LIN {X 0,Y 239.218,Z 1199.48,A -85,B 0,C 180,E1 5752.201,E2 5752.201} C_VEL
LIN {X 0,Y 256.307,Z 1187.286,A -85,B 0,C 180,E1 5754.218,E2 5754.218} C_VEL
LIN {X 0,Y 273.673,Z 1173.769,A -85,B 0,C 180,E1 5755.98,E2 5755.98} C_VEL
LIN {X 0,Y 294.221,Z 1156.22,A -85,B 0,C 180,E1 5757.756,E2 5757.756} C_VEL
LIN {X 0,Y 314.021,Z 1137.067,A -85,B 0,C 180,E1 5759.227,E2 5759.227} C_VEL
LIN {X 0,Y 329.492,Z 1120.573,A -85,B 0,C 180,E1 5760.229,E2 5760.229} C_VEL
LIN {X 0,Y 333.53,Z 1116.052,A -85,B 0,C 180,E1 5760.492,E2 5760.492} C_VEL
LIN {X 0,Y 325.823,Z 1124.556,A -85,B 0,C 180,E1 5761.006,E2 5761.006} C_VEL
LIN {X 0,Y 321.322,Z 1129.417,A -85,B 0,C 180,E1 5761.15,E2 5761.15} C_VEL
LIN {X 0,Y 315.113,Z 1135.776,A -85,B 0,C 180,E1 5760.961,E2 5760.961} C_VEL
LIN {X 0,Y 300.81,Z 1149.589,A -85,B 0,C 180,E1 5759.861,E2 5759.861} C_VEL
LIN {X 0,Y 283.612,Z 1164.923,A -85,B 0,C 180,E1 5758.586,E2 5758.586} C_VEL
LIN {X 0,Y 260.469,Z 1183.452,A -85,B 0,C 180,E1 5756.565,E2 5756.565} C_VEL
LIN {X 0,Y 240.904,Z 1197.395,A -85,B 0,C 180,E1 5754.522,E2 5754.522} C_VEL
LIN {X 0,Y 222.759,Z 1209.185,A -85,B 0,C 180,E1 5752.261,E2 5752.261} C_VEL
LIN {X 0,Y 204.429,Z 1220.07,A -85,B 0,C 180,E1 5749.508,E2 5749.508} C_VEL
LIN {X 0,Y 182.016,Z 1232.203,A -85,B 0,C 180,E1 5745.247,E2 5745.247} C_VEL
LIN {X 0,Y 160.819,Z 1242.295,A -85,B 0,C 180,E1 5739.896,E2 5739.896} C_VEL
LIN {X 0,Y 143.477,Z 1249.877,A -85,B 0,C 180,E1 5733.957,E2 5733.957} C_VEL
LIN {X 0,Y 128.105,Z 1256.155,A -85,B 0,C 180,E1 5726.665,E2 5726.665} C_VEL
LIN {X 0,Y 112.467,Z 1262.354,A -85,B 0,C 180,E1 5715.366,E2 5715.366} C_VEL
LIN {X 0,Y 101.995,Z 1266.473,A -85,B 0,C 180,E1 5701.992,E2 5701.992} C_VEL
LIN {X 0,Y 97.397,Z 1268.698,A -85,B 0,C 180,E1 5689.83,E2 5689.83} C_VEL
LIN {X 0,Y 96.077,Z 1269.823,A -85,B 0,C 180,E1 5678.405,E2 5678.405} C_VEL
LIN {X 0,Y 96.068,Z 1270.167,A -85,B 0,C 180,E1 5670.027,E2 5670.027} C_VEL
LIN {X 0,Y 96.076,Z 1269.821,A -85,B 0,C 180,E1 5661.65,E2 5661.65} C_VEL
LIN {X 0,Y 97.385,Z 1268.69,A -85,B 0,C 180,E1 5650.225,E2 5650.225} C_VEL
LIN {X 0,Y 102.276,Z 1266.336,A -85,B 0,C 180,E1 5637.505,E2 5637.505} C_VEL
LIN {X 0,Y 114.151,Z 1261.596,A -85,B 0,C 180,E1 5623.097,E2 5623.097} C_VEL
LIN {X 0,Y 128.042,Z 1256.122,A -85,B 0,C 180,E1 5613.367,E2 5613.367} C_VEL
LIN {X 0,Y 142.747,Z 1250.113,A -85,B 0,C 180,E1 5606.335,E2 5606.335} C_VEL
LIN {X 0,Y 159.123,Z 1242.966,A -85,B 0,C 180,E1 5600.603,E2 5600.603} C_VEL
LIN {X 0,Y 178.447,Z 1233.818,A -85,B 0,C 180,E1 5595.538,E2 5595.538} C_VEL
LIN {X 0,Y 202.513,Z 1221.049,A -85,B 0,C 180,E1 5590.808,E2 5590.808} C_VEL
LIN {X 0,Y 221.991,Z 1209.52,A -85,B 0,C 180,E1 5587.838,E2 5587.838} C_VEL
LIN {X 0,Y 240.822,Z 1197.285,A -85,B 0,C 180,E1 5585.48,E2 5585.48} C_VEL
LIN {X 0,Y 262.332,Z 1181.904,A -85,B 0,C 180,E1 5583.249,E2 5583.249} C_VEL
LIN {X 0,Y 283.988,Z 1164.363,A -85,B 0,C 180,E1 5581.374,E2 5581.374} C_VEL
LIN {X 0,Y 300.904,Z 1149.241,A -85,B 0,C 180,E1 5580.123,E2 5580.123} C_VEL
LIN {X 0,Y 311.366,Z 1139.22,A -85,B 0,C 180,E1 5579.418,E2 5579.418} C_VEL
LIN {X 0,Y 289.81,Z 1158.959,A -85,B 0,C 180,E1 5577.825,E2 5577.825} C_VEL
LIN {X 0,Y 272.462,Z 1173.195,A -85,B 0,C 180,E1 5576.347,E2 5576.347} C_VEL
LIN {X 0,Y 255.986,Z 1185.54,A -85,B 0,C 180,E1 5574.748,E2 5574.748} C_VEL
LIN {X 0,Y 238.263,Z 1197.663,A -85,B 0,C 180,E1 5572.767,E2 5572.767} C_VEL
LIN {X 0,Y 217.251,Z 1210.706,A -85,B 0,C 180,E1 5569.951,E2 5569.951} C_VEL
LIN {X 0,Y 194.579,Z 1223.116,A -85,B 0,C 180,E1 5566.15,E2 5566.15} C_VEL
LIN {X 0,Y 176.306,Z 1232.089,A -85,B 0,C 180,E1 5562.263,E2 5562.263} C_VEL
LIN {X 0,Y 158.961,Z 1239.833,A -85,B 0,C 180,E1 5557.565,E2 5557.565} C_VEL
LIN {X 0,Y 142.135,Z 1246.704,A -85,B 0,C 180,E1 5551.519,E2 5551.519} C_VEL
LIN {X 0,Y 123.389,Z 1253.713,A -85,B 0,C 180,E1 5541.779,E2 5541.779} C_VEL
LIN {X 0,Y 110.564,Z 1258.126,A -85,B 0,C 180,E1 5531.279,E2 5531.279} C_VEL
LIN {X 0,Y 102.223,Z 1261.043,A -85,B 0,C 180,E1 5519.893,E2 5519.893} C_VEL
LIN {X 0,Y 97.807,Z 1262.768,A -85,B 0,C 180,E1 5508.447,E2 5508.447} C_VEL
LIN {X 0,Y 96.278,Z 1263.591,A -85,B 0,C 180,E1 5497.731,E2 5497.731} C_VEL
LIN {X 0,Y 96.072,Z 1263.825,A -85,B 0,C 180,E1 5488.78,E2 5488.78} C_VEL
LIN {X 0,Y 96.5,Z 1263.503,A -85,B 0,C 180,E1 5479.224,E2 5479.224} C_VEL
LIN {X 0,Y 99.61,Z 1262.139,A -85,B 0,C 180,E1 5465.67,E2 5465.67} C_VEL
LIN {X 0,Y 107.516,Z 1259.227,A -85,B 0,C 180,E1 5452.107,E2 5452.107} C_VEL
LIN {X 0,Y 118.163,Z 1255.541,A -85,B 0,C 180,E1 5441.841,E2 5441.841} C_VEL
LIN {X 0,Y 130.982,Z 1250.967,A -85,B 0,C 180,E1 5433.656,E2 5433.656} C_VEL
LIN {X 0,Y 146.56,Z 1245.028,A -85,B 0,C 180,E1 5426.621,E2 5426.621} C_VEL
LIN {X 0,Y 167.103,Z 1236.5,A -85,B 0,C 180,E1 5420.007,E2 5420.007} C_VEL
LIN {X 0,Y 188.41,Z 1226.357,A -85,B 0,C 180,E1 5414.971,E2 5414.971} C_VEL
LIN {X 0,Y 207.193,Z 1216.475,A -85,B 0,C 180,E1 5411.532,E2 5411.532} C_VEL
LIN {X 0,Y 225.646,Z 1205.779,A -85,B 0,C 180,E1 5408.77,E2 5408.77} C_VEL
LIN {X 0,Y 248.133,Z 1191.364,A -85,B 0,C 180,E1 5406.014,E2 5406.014} C_VEL
LIN {X 0,Y 269.668,Z 1175.589,A -85,B 0,C 180,E1 5403.827,E2 5403.827} C_VEL
LIN {X 0,Y 286.244,Z 1162.22,A -85,B 0,C 180,E1 5402.382,E2 5402.382} C_VEL
LIN {X 0,Y 303.049,Z 1147.355,A -85,B 0,C 180,E1 5401.092,E2 5401.092} C_VEL
LIN {X 0,Y 310.756,Z 1140.13,A -85,B 0,C 180,E1 5400.53,E2 5400.53} C_VEL
LIN {X 0,Y 300.81,Z 1149.589,A -85,B 0,C 180,E1 5399.861,E2 5399.861} C_VEL
LIN {X 0,Y 295.137,Z 1154.893,A -85,B 0,C 180,E1 5399.66,E2 5399.66} C_VEL
LIN {X 0,Y 278.947,Z 1168.594,A -85,B 0,C 180,E1 5399.771,E2 5399.771} C_VEL
LIN {X 0,Y 273.814,Z 1172.595,A -85,B 0,C 180,E1 5399.544,E2 5399.544} C_VEL
LIN {X 0,Y 256.149,Z 1186.028,A -85,B 0,C 180,E1 5398.058,E2 5398.058} C_VEL
LIN {X 0,Y 238.493,Z 1198.284,A -85,B 0,C 180,E1 5396.336,E2 5396.336} C_VEL
LIN {X 0,Y 219.173,Z 1210.502,A -85,B 0,C 180,E1 5394.09,E2 5394.09} C_VEL
LIN {X 0,Y 195.602,Z 1223.934,A -85,B 0,C 180,E1 5390.668,E2 5390.668} C_VEL
LIN {X 0,Y 173.778,Z 1234.85,A -85,B 0,C 180,E1 5386.557,E2 5386.557} C_VEL
LIN {X 0,Y 155.3,Z 1243.23,A -85,B 0,C 180,E1 5381.998,E2 5381.998} C_VEL
LIN {X 0,Y 137.722,Z 1250.508,A -85,B 0,C 180,E1 5376.215,E2 5376.215} C_VEL
LIN {X 0,Y 118.244,Z 1257.965,A -85,B 0,C 180,E1 5366.877,E2 5366.877} C_VEL
LIN {X 0,Y 103.112,Z 1263.274,A -85,B 0,C 180,E1 5355.096,E2 5355.096} C_VEL
LIN {X 0,Y 94.07,Z 1266.568,A -85,B 0,C 180,E1 5342.857,E2 5342.857} C_VEL
LIN {X 0,Y 89.575,Z 1268.504,A -85,B 0,C 180,E1 5330.958,E2 5330.958} C_VEL
LIN {X 0,Y 88.096,Z 1269.562,A -85,B 0,C 180,E1 5319.084,E2 5319.084} C_VEL
LIN {X 0,Y 88.065,Z 1269.889,A -85,B 0,C 180,E1 5310.68,E2 5310.68} C_VEL
LIN {X 0,Y 88.074,Z 1269.61,A -85,B 0,C 180,E1 5302.2,E2 5302.2} C_VEL
LIN {X 0,Y 89.152,Z 1268.721,A -85,B 0,C 180,E1 5291.051,E2 5291.051} C_VEL
LIN {X 0,Y 93.127,Z 1266.92,A -85,B 0,C 180,E1 5279.013,E2 5279.013} C_VEL
LIN {X 0,Y 101.184,Z 1263.918,A -85,B 0,C 180,E1 5266.992,E2 5266.992} C_VEL
LIN {X 0,Y 113.098,Z 1259.676,A -85,B 0,C 180,E1 5256.479,E2 5256.479} C_VEL
LIN {X 0,Y 128.614,Z 1253.989,A -85,B 0,C 180,E1 5247.641,E2 5247.641} C_VEL
LIN {X 0,Y 151.313,Z 1244.882,A -85,B 0,C 180,E1 5239.161,E2 5239.161} C_VEL
LIN {X 0,Y 170.149,Z 1236.454,A -85,B 0,C 180,E1 5234.233,E2 5234.233} C_VEL
LIN {X 0,Y 188.136,Z 1227.63,A -85,B 0,C 180,E1 5230.605,E2 5230.605} C_VEL
LIN {X 0,Y 206.734,Z 1217.61,A -85,B 0,C 180,E1 5227.597,E2 5227.597} C_VEL
LIN {X 0,Y 229.667,Z 1203.974,A -85,B 0,C 180,E1 5224.637,E2 5224.637} C_VEL
LIN {X 0,Y 252.115,Z 1188.752,A -85,B 0,C 180,E1 5222.304,E2 5222.304} C_VEL
LIN {X 0,Y 269.932,Z 1175.428,A -85,B 0,C 180,E1 5220.751,E2 5220.751} C_VEL
LIN {X 0,Y 286.918,Z 1161.515,A -85,B 0,C 180,E1 5219.471,E2 5219.471} C_VEL
LIN {X 0,Y 288.401,Z 1160.248,A -85,B 0,C 180,E1 5219.367,E2 5219.367} C_VEL
LIN {X 0,Y 271.073,Z 1174.227,A -85,B 0,C 180,E1 5218.002,E2 5218.002} C_VEL
LIN {X 0,Y 253.408,Z 1187.192,A -85,B 0,C 180,E1 5216.413,E2 5216.413} C_VEL
LIN {X 0,Y 232.122,Z 1201.336,A -85,B 0,C 180,E1 5214.155,E2 5214.155} C_VEL
LIN {X 0,Y 208.446,Z 1215.124,A -85,B 0,C 180,E1 5211.069,E2 5211.069} C_VEL
LIN {X 0,Y 190.022,Z 1224.734,A -85,B 0,C 180,E1 5208.077,E2 5208.077} C_VEL
LIN {X 0,Y 172.194,Z 1233.152,A -85,B 0,C 180,E1 5204.493,E2 5204.493} C_VEL
LIN {X 0,Y 153.483,Z 1241.135,A -85,B 0,C 180,E1 5199.678,E2 5199.678} C_VEL
LIN {X 0,Y 131.593,Z 1249.466,A -85,B 0,C 180,E1 5191.764,E2 5191.764} C_VEL
LIN {X 0,Y 115.247,Z 1254.97,A -85,B 0,C 180,E1 5182.916,E2 5182.916} C_VEL
LIN {X 0,Y 103.502,Z 1258.699,A -85,B 0,C 180,E1 5173.268,E2 5173.268} C_VEL
LIN {X 0,Y 94.868,Z 1261.418,A -85,B 0,C 180,E1 5161.768,E2 5161.768} C_VEL
LIN {X 0,Y 89.971,Z 1263.097,A -85,B 0,C 180,E1 5149.444,E2 5149.444} C_VEL
LIN {X 0,Y 88.322,Z 1263.854,A -85,B 0,C 180,E1 5138.433,E2 5138.433} C_VEL
LIN {X 0,Y 88.078,Z 1264.087,A -85,B 0,C 180,E1 5128.669,E2 5128.669} C_VEL
LIN {X 0,Y 88.591,Z 1263.768,A -85,B 0,C 180,E1 5118.249,E2 5118.249} C_VEL
LIN {X 0,Y 92.226,Z 1262.407,A -85,B 0,C 180,E1 5103.578,E2 5103.578} C_VEL
LIN {X 0,Y 101.128,Z 1259.498,A -85,B 0,C 180,E1 5089.233,E2 5089.233} C_VEL
LIN {X 0,Y 112.795,Z 1255.813,A -85,B 0,C 180,E1 5078.699,E2 5078.699} C_VEL
LIN {X 0,Y 126.554,Z 1251.24,A -85,B 0,C 180,E1 5070.514,E2 5070.514} C_VEL
LIN {X 0,Y 142.232,Z 1245.594,A -85,B 0,C 180,E1 5063.912,E2 5063.912} C_VEL
LIN {X 0,Y 161.421,Z 1237.984,A -85,B 0,C 180,E1 5058.042,E2 5058.042} C_VEL
LIN {X 0,Y 185.529,Z 1227.076,A -85,B 0,C 180,E1 5052.664,E2 5052.664} C_VEL
LIN {X 0,Y 204.759,Z 1217.25,A -85,B 0,C 180,E1 5049.397,E2 5049.397} C_VEL
LIN {X 0,Y 223.576,Z 1206.612,A -85,B 0,C 180,E1 5046.79,E2 5046.79} C_VEL
LIN {X 0,Y 243.791,Z 1193.966,A -85,B 0,C 180,E1 5044.469,E2 5044.469} C_VEL
LIN {X 0,Y 267.205,Z 1177.426,A -85,B 0,C 180,E1 5042.245,E2 5042.245} C_VEL
LIN {X 0,Y 285.045,Z 1163.305,A -85,B 0,C 180,E1 5040.804,E2 5040.804} C_VEL
LIN {X 0,Y 287.787,Z 1161.011,A -85,B 0,C 180,E1 5040.581,E2 5040.581} C_VEL
LIN {X 0,Y 273.814,Z 1172.595,A -85,B 0,C 180,E1 5039.544,E2 5039.544} C_VEL
LIN {X 0,Y 267.746,Z 1177.324,A -85,B 0,C 180,E1 5039.286,E2 5039.286} C_VEL
LIN {X 0,Y 250.57,Z 1189.79,A -85,B 0,C 180,E1 5039.298,E2 5039.298} C_VEL
LIN {X 0,Y 245.141,Z 1193.419,A -85,B 0,C 180,E1 5039.007,E2 5039.007} C_VEL
LIN {X 0,Y 223.347,Z 1207.302,A -85,B 0,C 180,E1 5036.843,E2 5036.843} C_VEL
LIN {X 0,Y 203.956,Z 1218.465,A -85,B 0,C 180,E1 5034.484,E2 5034.484} C_VEL
LIN {X 0,Y 184.042,Z 1228.835,A -85,B 0,C 180,E1 5031.488,E2 5031.488} C_VEL
LIN {X 0,Y 160.251,Z 1239.918,A -85,B 0,C 180,E1 5026.804,E2 5026.804} C_VEL
LIN {X 0,Y 138.659,Z 1248.66,A -85,B 0,C 180,E1 5020.898,E2 5020.898} C_VEL
LIN {X 0,Y 121.937,Z 1254.809,A -85,B 0,C 180,E1 5014.466,E2 5014.466} C_VEL
LIN {X 0,Y 106.408,Z 1260.079,A -85,B 0,C 180,E1 5005.822,E2 5005.822} C_VEL
LIN {X 0,Y 92.761,Z 1264.525,A -85,B 0,C 180,E1 4993.655,E2 4993.655} C_VEL
LIN {X 0,Y 83.032,Z 1267.858,A -85,B 0,C 180,E1 4976.493,E2 4976.493} C_VEL
LIN {X 0,Y 80.19,Z 1269.237,A -85,B 0,C 180,E1 4961.54,E2 4961.54} C_VEL
LIN {X 0,Y 80.077,Z 1269.58,A -85,B 0,C 180,E1 4952.179,E2 4952.179} C_VEL
LIN {X 0,Y 80.072,Z 1269.426,A -85,B 0,C 180,E1 4943.58,E2 4943.58} C_VEL
LIN {X 0,Y 81.04,Z 1268.677,A -85,B 0,C 180,E1 4931.324,E2 4931.324} C_VEL
LIN {X 0,Y 85.807,Z 1266.771,A -85,B 0,C 180,E1 4916.831,E2 4916.831} C_VEL
LIN {X 0,Y 95.211,Z 1263.656,A -85,B 0,C 180,E1 4903.606,E2 4903.606} C_VEL
LIN {X 0,Y 108.003,Z 1259.502,A -85,B 0,C 180,E1 4893.108,E2 4893.108} C_VEL
LIN {X 0,Y 124.154,Z 1253.976,A -85,B 0,C 180,E1 4884.544,E2 4884.544} C_VEL
LIN {X 0,Y 147.032,Z 1245.333,A -85,B 0,C 180,E1 4876.564,E2 4876.564} C_VEL
LIN {X 0,Y 168.272,Z 1236.176,A -85,B 0,C 180,E1 4871.444,E2 4871.444} C_VEL
LIN {X 0,Y 187.226,Z 1227.121,A -85,B 0,C 180,E1 4867.982,E2 4867.982} C_VEL
LIN {X 0,Y 206.752,Z 1216.805,A -85,B 0,C 180,E1 4865.143,E2 4865.143} C_VEL
LIN {X 0,Y 231.107,Z 1202.429,A -85,B 0,C 180,E1 4862.336,E2 4862.336} C_VEL
LIN {X 0,Y 251.918,Z 1188.475,A -85,B 0,C 180,E1 4860.398,E2 4860.398} C_VEL
LIN {X 0,Y 265.344,Z 1178.737,A -85,B 0,C 180,E1 4859.318,E2 4859.318} C_VEL
LIN {X 0,Y 242.183,Z 1194.755,A -85,B 0,C 180,E1 4857.295,E2 4857.295} C_VEL
LIN {X 0,Y 222.682,Z 1206.763,A -85,B 0,C 180,E1 4855.247,E2 4855.247} C_VEL
LIN {X 0,Y 204.462,Z 1216.909,A -85,B 0,C 180,E1 4852.958,E2 4852.958} C_VEL
LIN {X 0,Y 185.529,Z 1226.429,A -85,B 0,C 180,E1 4850.069,E2 4850.069} C_VEL
LIN {X 0,Y 162.12,Z 1236.957,A -85,B 0,C 180,E1 4845.46,E2 4845.46} C_VEL
LIN {X 0,Y 139.87,Z 1245.497,A -85,B 0,C 180,E1 4839.407,E2 4839.407} C_VEL
LIN {X 0,Y 122.753,Z 1251.375,A -85,B 0,C 180,E1 4832.861,E2 4832.861} C_VEL
LIN {X 0,Y 107.802,Z 1256.031,A -85,B 0,C 180,E1 4824.662,E2 4824.662} C_VEL
LIN {X 0,Y 94.535,Z 1259.876,A -85,B 0,C 180,E1 4813.391,E2 4813.391} C_VEL
LIN {X 0,Y 84.155,Z 1262.872,A -85,B 0,C 180,E1 4796.803,E2 4796.803} C_VEL
LIN {X 0,Y 80.543,Z 1264.063,A -85,B 0,C 180,E1 4781.423,E2 4781.423} C_VEL
LIN {X 0,Y 80.08,Z 1264.366,A -85,B 0,C 180,E1 4770.683,E2 4770.683} C_VEL
LIN {X 0,Y 80.422,Z 1264.106,A -85,B 0,C 180,E1 4759.943,E2 4759.943} C_VEL
LIN {X 0,Y 83.18,Z 1263.135,A -85,B 0,C 180,E1 4745.844,E2 4745.844} C_VEL
LIN {X 0,Y 92.158,Z 1260.661,A -85,B 0,C 180,E1 4729.35,E2 4729.35} C_VEL
LIN {X 0,Y 106.516,Z 1256.478,A -85,B 0,C 180,E1 4716.13,E2 4716.13} C_VEL
LIN {X 0,Y 121.787,Z 1251.757,A -85,B 0,C 180,E1 4707.499,E2 4707.499} C_VEL
LIN {X 0,Y 138.241,Z 1246.159,A -85,B 0,C 180,E1 4701.041,E2 4701.041} C_VEL
LIN {X 0,Y 156.875,Z 1239.1,A -85,B 0,C 180,E1 4695.704,E2 4695.704} C_VEL
LIN {X 0,Y 180.195,Z 1229.14,A -85,B 0,C 180,E1 4690.778,E2 4690.778} C_VEL
LIN {X 0,Y 202.616,Z 1218.025,A -85,B 0,C 180,E1 4687.215,E2 4687.215} C_VEL
LIN {X 0,Y 221.778,Z 1207.445,A -85,B 0,C 180,E1 4684.776,E2 4684.776} C_VEL
LIN {X 0,Y 240.293,Z 1196.135,A -85,B 0,C 180,E1 4682.806,E2 4682.806} C_VEL
LIN {X 0,Y 262.031,Z 1181.414,A -85,B 0,C 180,E1 4680.87,E2 4680.87} C_VEL
LIN {X 0,Y 264.69,Z 1179.465,A -85,B 0,C 180,E1 4680.623,E2 4680.623} C_VEL
LIN {X 0,Y 245.141,Z 1193.419,A -85,B 0,C 180,E1 4679.007,E2 4679.007} C_VEL
LIN {X 0,Y 238.694,Z 1197.621,A -85,B 0,C 180,E1 4678.671,E2 4678.671} C_VEL
LIN {X 0,Y 221.471,Z 1208.041,A -85,B 0,C 180,E1 4678.58,E2 4678.58} C_VEL
LIN {X 0,Y 214.936,Z 1211.815,A -85,B 0,C 180,E1 4678.17,E2 4678.17} C_VEL
LIN {X 0,Y 189.712,Z 1225.265,A -85,B 0,C 180,E1 4675.083,E2 4675.083} C_VEL
LIN {X 0,Y 169.313,Z 1234.887,A -85,B 0,C 180,E1 4671.852,E2 4671.852} C_VEL
LIN {X 0,Y 150.321,Z 1242.925,A -85,B 0,C 180,E1 4667.972,E2 4667.972} C_VEL
LIN {X 0,Y 130.114,Z 1250.584,A -85,B 0,C 180,E1 4662.401,E2 4662.401} C_VEL
LIN {X 0,Y 106.963,Z 1258.283,A -85,B 0,C 180,E1 4652.677,E2 4652.677} C_VEL
LIN {X 0,Y 91.468,Z 1262.896,A -85,B 0,C 180,E1 4641.955,E2 4641.955} C_VEL
LIN {X 0,Y 80.658,Z 1266.025,A -85,B 0,C 180,E1 4629.254,E2 4629.254} C_VEL
LIN {X 0,Y 74.492,Z 1267.966,A -85,B 0,C 180,E1 4615.475,E2 4615.475} C_VEL
LIN {X 0,Y 72.171,Z 1269.027,A -85,B 0,C 180,E1 4601.22,E2 4601.22} C_VEL
LIN {X 0,Y 72.073,Z 1269.364,A -85,B 0,C 180,E1 4590.831,E2 4590.831} C_VEL
LIN {X 0,Y 72.091,Z 1269.108,A -85,B 0,C 180,E1 4581.261,E2 4581.261} C_VEL
LIN {X 0,Y 73.508,Z 1268.334,A -85,B 0,C 180,E1 4568.493,E2 4568.493} C_VEL
LIN {X 0,Y 79.011,Z 1266.499,A -85,B 0,C 180,E1 4553.546,E2 4553.546} C_VEL
LIN {X 0,Y 89.081,Z 1263.551,A -85,B 0,C 180,E1 4540.296,E2 4540.296} C_VEL
LIN {X 0,Y 102.765,Z 1259.496,A -85,B 0,C 180,E1 4529.75,E2 4529.75} C_VEL
LIN {X 0,Y 119.275,Z 1254.229,A -85,B 0,C 180,E1 4521.552,E2 4521.552} C_VEL
LIN {X 0,Y 139.542,Z 1247.078,A -85,B 0,C 180,E1 4514.769,E2 4514.769} C_VEL
LIN {X 0,Y 164.012,Z 1237.142,A -85,B 0,C 180,E1 4509.12,E2 4509.12} C_VEL
LIN {X 0,Y 184.81,Z 1227.543,A -85,B 0,C 180,E1 4505.615,E2 4505.615} C_VEL
LIN {X 0,Y 204.207,Z 1217.579,A -85,B 0,C 180,E1 4503.038,E2 4503.038} C_VEL
LIN {X 0,Y 224.939,Z 1205.758,A -85,B 0,C 180,E1 4500.808,E2 4500.808} C_VEL
LIN {X 0,Y 241.934,Z 1195.029,A -85,B 0,C 180,E1 4499.256,E2 4499.256} C_VEL
LIN {X 0,Y 222.148,Z 1207.038,A -85,B 0,C 180,E1 4497.383,E2 4497.383} C_VEL
LIN {X 0,Y 202.872,Z 1217.567,A -85,B 0,C 180,E1 4495.194,E2 4495.194} C_VEL
LIN {X 0,Y 182.546,Z 1227.521,A -85,B 0,C 180,E1 4492.356,E2 4492.356} C_VEL
LIN {X 0,Y 156.592,Z 1238.604,A -85,B 0,C 180,E1 4487.581,E2 4487.581} C_VEL
LIN {X 0,Y 136.301,Z 1246.065,A -85,B 0,C 180,E1 4482.416,E2 4482.416} C_VEL
LIN {X 0,Y 118.945,Z 1251.723,A -85,B 0,C 180,E1 4476.327,E2 4476.327} C_VEL
LIN {X 0,Y 102.528,Z 1256.501,A -85,B 0,C 180,E1 4467.991,E2 4467.991} C_VEL
LIN {X 0,Y 86.069,Z 1260.896,A -85,B 0,C 180,E1 4454.144,E2 4454.144} C_VEL
LIN {X 0,Y 75.812,Z 1263.385,A -85,B 0,C 180,E1 4436.603,E2 4436.603} C_VEL
LIN {X 0,Y 72.495,Z 1264.365,A -85,B 0,C 180,E1 4421.096,E2 4421.096} C_VEL
LIN {X 0,Y 72.088,Z 1264.647,A -85,B 0,C 180,E1 4409.964,E2 4409.964} C_VEL
LIN {X 0,Y 72.577,Z 1264.352,A -85,B 0,C 180,E1 4398.038,E2 4398.038} C_VEL
LIN {X 0,Y 76.357,Z 1263.281,A -85,B 0,C 180,E1 4381.837,E2 4381.837} C_VEL
LIN {X 0,Y 87.632,Z 1260.492,A -85,B 0,C 180,E1 4364.002,E2 4364.002} C_VEL
LIN {X 0,Y 102.534,Z 1256.553,A -85,B 0,C 180,E1 4351.919,E2 4351.919} C_VEL
LIN {X 0,Y 118.962,Z 1251.785,A -85,B 0,C 180,E1 4343.582,E2 4343.582} C_VEL
LIN {X 0,Y 136.327,Z 1246.139,A -85,B 0,C 180,E1 4337.491,E2 4337.491} C_VEL
LIN {X 0,Y 156.629,Z 1238.689,A -85,B 0,C 180,E1 4332.324,E2 4332.324} C_VEL
LIN {X 0,Y 182.615,Z 1227.613,A -85,B 0,C 180,E1 4327.551,E2 4327.551} C_VEL
LIN {X 0,Y 202.706,Z 1217.794,A -85,B 0,C 180,E1 4324.745,E2 4324.745} C_VEL
LIN {X 0,Y 221.668,Z 1207.472,A -85,B 0,C 180,E1 4322.585,E2 4322.585} C_VEL
LIN {X 0,Y 241.575,Z 1195.438,A -85,B 0,C 180,E1 4320.682,E2 4320.682} C_VEL
LIN {X 0,Y 222.049,Z 1207.612,A -85,B 0,C 180,E1 4318.905,E2 4318.905} C_VEL
LIN {X 0,Y 214.936,Z 1211.815,A -85,B 0,C 180,E1 4318.17,E2 4318.17} C_VEL
LIN {X 0,Y 208.32,Z 1215.528,A -85,B 0,C 180,E1 4317.725,E2 4317.725} C_VEL
LIN {X 0,Y 190.307,Z 1224.513,A -85,B 0,C 180,E1 4317.451,E2 4317.451} C_VEL
LIN {X 0,Y 183.482,Z 1227.718,A -85,B 0,C 180,E1 4316.905,E2 4316.905} C_VEL
LIN {X 0,Y 159.036,Z 1238.656,A -85,B 0,C 180,E1 4313.139,E2 4313.139} C_VEL
LIN {X 0,Y 134.99,Z 1247.794,A -85,B 0,C 180,E1 4307.966,E2 4307.966} C_VEL
LIN {X 0,Y 115.673,Z 1254.257,A -85,B 0,C 180,E1 4302.024,E2 4302.024} C_VEL
LIN {X 0,Y 97.915,Z 1259.542,A -85,B 0,C 180,E1 4293.953,E2 4293.953} C_VEL
LIN {X 0,Y 81.514,Z 1263.979,A -85,B 0,C 180,E1 4281.774,E2 4281.774} C_VEL
LIN {X 0,Y 68.368,Z 1267.394,A -85,B 0,C 180,E1 4261.812,E2 4261.812} C_VEL
LIN {X 0,Y 64.312,Z 1268.734,A -85,B 0,C 180,E1 4243.527,E2 4243.527} C_VEL
LIN {X 0,Y 64.081,Z 1269.078,A -85,B 0,C 180,E1 4231.829,E2 4231.829} C_VEL
LIN {X 0,Y 64.086,Z 1268.897,A -85,B 0,C 180,E1 4221.969,E2 4221.969} C_VEL
LIN {X 0,Y 65.757,Z 1268.14,A -85,B 0,C 180,E1 4206.757,E2 4206.757} C_VEL
LIN {X 0,Y 72.524,Z 1266.227,A -85,B 0,C 180,E1 4189.66,E2 4189.66} C_VEL
LIN {X 0,Y 83.916,Z 1263.276,A -85,B 0,C 180,E1 4175.938,E2 4175.938} C_VEL
LIN {X 0,Y 98.647,Z 1259.28,A -85,B 0,C 180,E1 4165.632,E2 4165.632} C_VEL
LIN {X 0,Y 116.442,Z 1253.952,A -85,B 0,C 180,E1 4157.691,E2 4157.691} C_VEL
LIN {X 0,Y 138.54,Z 1246.484,A -85,B 0,C 180,E1 4151.137,E2 4151.137} C_VEL
LIN {X 0,Y 163.832,Z 1236.452,A -85,B 0,C 180,E1 4146.027,E2 4146.027} C_VEL
LIN {X 0,Y 184.175,Z 1227.264,A -85,B 0,C 180,E1 4142.998,E2 4142.998} C_VEL
LIN {X 0,Y 203.934,Z 1217.301,A -85,B 0,C 180,E1 4140.671,E2 4140.671} C_VEL
LIN {X 0,Y 218.555,Z 1209.213,A -85,B 0,C 180,E1 4139.214,E2 4139.214} C_VEL
LIN {X 0,Y 194.263,Z 1221.977,A -85,B 0,C 180,E1 4136.604,E2 4136.604} C_VEL
LIN {X 0,Y 170.019,Z 1232.831,A -85,B 0,C 180,E1 4133.245,E2 4133.245} C_VEL
LIN {X 0,Y 150.337,Z 1240.602,A -85,B 0,C 180,E1 4129.655,E2 4129.655} C_VEL
LIN {X 0,Y 130.801,Z 1247.4,A -85,B 0,C 180,E1 4124.935,E2 4124.935} C_VEL
LIN {X 0,Y 108.487,Z 1254.194,A -85,B 0,C 180,E1 4117.101,E2 4117.101} C_VEL
LIN {X 0,Y 88.46,Z 1259.213,A -85,B 0,C 180,E1 4105.545,E2 4105.545} C_VEL
LIN {X 0,Y 75.54,Z 1262.122,A -85,B 0,C 180,E1 4092.409,E2 4092.409} C_VEL
LIN {X 0,Y 67.725,Z 1263.837,A -85,B 0,C 180,E1 4077.193,E2 4077.193} C_VEL
LIN {X 0,Y 64.521,Z 1264.648,A -85,B 0,C 180,E1 4061.58,E2 4061.58} C_VEL
LIN {X 0,Y 64.087,Z 1264.897,A -85,B 0,C 180,E1 4049.065,E2 4049.065} C_VEL
LIN {X 0,Y 64.708,Z 1264.617,A -85,B 0,C 180,E1 4036.557,E2 4036.557} C_VEL
LIN {X 0,Y 69.507,Z 1263.505,A -85,B 0,C 180,E1 4018.075,E2 4018.075} C_VEL
LIN {X 0,Y 82.712,Z 1260.611,A -85,B 0,C 180,E1 3999.269,E2 3999.269} C_VEL
LIN {X 0,Y 99.15,Z 1256.628,A -85,B 0,C 180,E1 3987.396,E2 3987.396} C_VEL
LIN {X 0,Y 116.606,Z 1251.847,A -85,B 0,C 180,E1 3979.538,E2 3979.538} C_VEL
LIN {X 0,Y 135.839,Z 1245.828,A -85,B 0,C 180,E1 3973.612,E2 3973.612} C_VEL
LIN {X 0,Y 160.687,Z 1236.827,A -85,B 0,C 180,E1 3968.265,E2 3968.265} C_VEL
LIN {X 0,Y 183.627,Z 1226.998,A -85,B 0,C 180,E1 3964.679,E2 3964.679} C_VEL
LIN {X 0,Y 203.424,Z 1217.433,A -85,B 0,C 180,E1 3962.254,E2 3962.254} C_VEL
LIN {X 0,Y 218.026,Z 1209.677,A -85,B 0,C 180,E1 3960.718,E2 3960.718} C_VEL
LIN {X 0,Y 193.118,Z 1223.106,A -85,B 0,C 180,E1 3958.114,E2 3958.114} C_VEL
LIN {X 0,Y 183.482,Z 1227.718,A -85,B 0,C 180,E1 3956.905,E2 3956.905} C_VEL
LIN {X 0,Y 176.63,Z 1230.952,A -85,B 0,C 180,E1 3956.312,E2 3956.312} C_VEL
LIN {X 0,Y 157.014,Z 1238.913,A -85,B 0,C 180,E1 3955.695,E2 3955.695} C_VEL
LIN {X 0,Y 151.04,Z 1241.115,A -85,B 0,C 180,E1 3954.998,E2 3954.998} C_VEL
LIN {X 0,Y 130.68,Z 1248.46,A -85,B 0,C 180,E1 3950.87,E2 3950.87} C_VEL
LIN {X 0,Y 110.7,Z 1254.777,A -85,B 0,C 180,E1 3945.2,E2 3945.2} C_VEL
LIN {X 0,Y 88.233,Z 1260.983,A -85,B 0,C 180,E1 3935.101,E2 3935.101} C_VEL
LIN {X 0,Y 70.318,Z 1265.112,A -85,B 0,C 180,E1 3920.216,E2 3920.216} C_VEL
LIN {X 0,Y 60.431,Z 1267.352,A -85,B 0,C 180,E1 3903.144,E2 3903.144} C_VEL
LIN {X 0,Y 56.366,Z 1268.496,A -85,B 0,C 180,E1 3884.427,E2 3884.427} C_VEL
LIN {X 0,Y 56.084,Z 1268.816,A -85,B 0,C 180,E1 3872.09,E2 3872.09} C_VEL
LIN {X 0,Y 56.09,Z 1268.659,A -85,B 0,C 180,E1 3861.849,E2 3861.849} C_VEL
LIN {X 0,Y 58.081,Z 1267.947,A -85,B 0,C 180,E1 3844.56,E2 3844.56} C_VEL
LIN {X 0,Y 66.42,Z 1265.954,A -85,B 0,C 180,E1 3825.024,E2 3825.024} C_VEL
LIN {X 0,Y 79.298,Z 1263.001,A -85,B 0,C 180,E1 3811.04,E2 3811.04} C_VEL
LIN {X 0,Y 95.309,Z 1259.004,A -85,B 0,C 180,E1 3801.067,E2 3801.067} C_VEL
LIN {X 0,Y 114.162,Z 1253.674,A -85,B 0,C 180,E1 3793.655,E2 3793.655} C_VEL
LIN {X 0,Y 137.158,Z 1246.206,A -85,B 0,C 180,E1 3787.669,E2 3787.669} C_VEL
LIN {X 0,Y 163.161,Z 1236.173,A -85,B 0,C 180,E1 3783.072,E2 3783.072} C_VEL
LIN {X 0,Y 184.409,Z 1226.758,A -85,B 0,C 180,E1 3780.311,E2 3780.311} C_VEL
LIN {X 0,Y 194.942,Z 1221.76,A -85,B 0,C 180,E1 3779.166,E2 3779.166} C_VEL
LIN {X 0,Y 170.3,Z 1232.678,A -85,B 0,C 180,E1 3776.199,E2 3776.199} C_VEL
LIN {X 0,Y 150.049,Z 1240.523,A -85,B 0,C 180,E1 3772.995,E2 3772.995} C_VEL
LIN {X 0,Y 130.377,Z 1247.2,A -85,B 0,C 180,E1 3768.888,E2 3768.888} C_VEL
LIN {X 0,Y 110.673,Z 1253.004,A -85,B 0,C 180,E1 3763.177,E2 3763.177} C_VEL
LIN {X 0,Y 88.525,Z 1258.583,A -85,B 0,C 180,E1 3753.092,E2 3753.092} C_VEL
LIN {X 0,Y 70.834,Z 1262.182,A -85,B 0,C 180,E1 3738.371,E2 3738.371} C_VEL
LIN {X 0,Y 60.925,Z 1264.043,A -85,B 0,C 180,E1 3721.628,E2 3721.628} C_VEL
LIN {X 0,Y 56.764,Z 1264.894,A -85,B 0,C 180,E1 3704.228,E2 3704.228} C_VEL
LIN {X 0,Y 56.096,Z 1265.172,A -85,B 0,C 180,E1 3689.953,E2 3689.953} C_VEL
LIN {X 0,Y 56.772,Z 1264.899,A -85,B 0,C 180,E1 3675.624,E2 3675.624} C_VEL
LIN {X 0,Y 61.284,Z 1264,A -85,B 0,C 180,E1 3657.376,E2 3657.376} C_VEL
LIN {X 0,Y 72.031,Z 1262,A -85,B 0,C 180,E1 3640.176,E2 3640.176} C_VEL
LIN {X 0,Y 92.424,Z 1257.688,A -85,B 0,C 180,E1 3624.606,E2 3624.606} C_VEL
LIN {X 0,Y 112.455,Z 1252.575,A -85,B 0,C 180,E1 3616.131,E2 3616.131} C_VEL
LIN {X 0,Y 131.347,Z 1246.978,A -85,B 0,C 180,E1 3610.792,E2 3610.792} C_VEL
LIN {X 0,Y 152.018,Z 1239.92,A -85,B 0,C 180,E1 3606.568,E2 3606.568} C_VEL
LIN {X 0,Y 177.229,Z 1229.956,A -85,B 0,C 180,E1 3602.81,E2 3602.81} C_VEL
LIN {X 0,Y 194.619,Z 1222.067,A -85,B 0,C 180,E1 3600.783,E2 3600.783} C_VEL
LIN {X 0,Y 169.144,Z 1233.745,A -85,B 0,C 180,E1 3597.778,E2 3597.778} C_VEL
LIN {X 0,Y 151.04,Z 1241.115,A -85,B 0,C 180,E1 3594.998,E2 3594.998} C_VEL
LIN {X 0,Y 144.033,Z 1243.708,A -85,B 0,C 180,E1 3594.154,E2 3594.154} C_VEL
LIN {X 0,Y 123.972,Z 1250.165,A -85,B 0,C 180,E1 3592.987,E2 3592.987} C_VEL
LIN {X 0,Y 117.924,Z 1251.916,A -85,B 0,C 180,E1 3591.955,E2 3591.955} C_VEL
LIN {X 0,Y 95.324,Z 1258.109,A -85,B 0,C 180,E1 3584.894,E2 3584.894} C_VEL
LIN {X 0,Y 77.734,Z 1262.243,A -85,B 0,C 180,E1 3576.036,E2 3576.036} C_VEL
LIN {X 0,Y 62.716,Z 1265.331,A -85,B 0,C 180,E1 3562.924,E2 3562.924} C_VEL
LIN {X 0,Y 52.528,Z 1267.31,A -85,B 0,C 180,E1 3544.883,E2 3544.883} C_VEL
LIN {X 0,Y 48.437,Z 1268.258,A -85,B 0,C 180,E1 3525.622,E2 3525.622} C_VEL
LIN {X 0,Y 48.085,Z 1268.577,A -85,B 0,C 180,E1 3511.246,E2 3511.246} C_VEL
LIN {X 0,Y 48.143,Z 1268.367,A -85,B 0,C 180,E1 3499.283,E2 3499.283} C_VEL
LIN {X 0,Y 51.148,Z 1267.591,A -85,B 0,C 180,E1 3479.334,E2 3479.334} C_VEL
LIN {X 0,Y 60.827,Z 1265.681,A -85,B 0,C 180,E1 3459.484,E2 3459.484} C_VEL
LIN {X 0,Y 75.325,Z 1262.726,A -85,B 0,C 180,E1 3445.579,E2 3445.579} C_VEL
LIN {X 0,Y 92.619,Z 1258.727,A -85,B 0,C 180,E1 3436.204,E2 3436.204} C_VEL
LIN {X 0,Y 112.468,Z 1253.396,A -85,B 0,C 180,E1 3429.47,E2 3429.47} C_VEL
LIN {X 0,Y 136.288,Z 1245.927,A -85,B 0,C 180,E1 3424.144,E2 3424.144} C_VEL
LIN {X 0,Y 162.927,Z 1235.893,A -85,B 0,C 180,E1 3420.098,E2 3420.098} C_VEL
LIN {X 0,Y 170.945,Z 1232.559,A -85,B 0,C 180,E1 3419.122,E2 3419.122} C_VEL
LIN {X 0,Y 149.111,Z 1240.851,A -85,B 0,C 180,E1 3416.155,E2 3416.155} C_VEL
LIN {X 0,Y 128.372,Z 1247.677,A -85,B 0,C 180,E1 3412.391,E2 3412.391} C_VEL
LIN {X 0,Y 106.745,Z 1253.766,A -85,B 0,C 180,E1 3406.829,E2 3406.829} C_VEL
LIN {X 0,Y 81.602,Z 1259.503,A -85,B 0,C 180,E1 3396.149,E2 3396.149} C_VEL
LIN {X 0,Y 65.001,Z 1262.558,A -85,B 0,C 180,E1 3383.049,E2 3383.049} C_VEL
LIN {X 0,Y 54.141,Z 1264.312,A -85,B 0,C 180,E1 3366.165,E2 3366.165} C_VEL
LIN {X 0,Y 48.928,Z 1265.165,A -85,B 0,C 180,E1 3346.159,E2 3346.159} C_VEL
LIN {X 0,Y 48.099,Z 1265.434,A -85,B 0,C 180,E1 3329.946,E2 3329.946} C_VEL
LIN {X 0,Y 48.911,Z 1265.173,A -85,B 0,C 180,E1 3313.91,E2 3313.91} C_VEL
LIN {X 0,Y 54.153,Z 1264.329,A -85,B 0,C 180,E1 3293.725,E2 3293.725} C_VEL
LIN {X 0,Y 65.677,Z 1262.481,A -85,B 0,C 180,E1 3276.145,E2 3276.145} C_VEL
LIN {X 0,Y 85.952,Z 1258.739,A -85,B 0,C 180,E1 3261.39,E2 3261.39} C_VEL
LIN {X 0,Y 109.518,Z 1253.091,A -85,B 0,C 180,E1 3252.243,E2 3252.243} C_VEL
LIN {X 0,Y 130.042,Z 1247.251,A -85,B 0,C 180,E1 3247.173,E2 3247.173} C_VEL
LIN {X 0,Y 151.416,Z 1240.148,A -85,B 0,C 180,E1 3243.407,E2 3243.407} C_VEL
LIN {X 0,Y 170.622,Z 1232.807,A -85,B 0,C 180,E1 3240.829,E2 3240.829} C_VEL
LIN {X 0,Y 149.112,Z 1241.365,A -85,B 0,C 180,E1 3237.993,E2 3237.993} C_VEL
LIN {X 0,Y 128.645,Z 1248.498,A -85,B 0,C 180,E1 3234.366,E2 3234.366} C_VEL
LIN {X 0,Y 117.924,Z 1251.916,A -85,B 0,C 180,E1 3231.955,E2 3231.955} C_VEL
LIN {X 0,Y 110.839,Z 1253.884,A -85,B 0,C 180,E1 3230.667,E2 3230.667} C_VEL
LIN {X 0,Y 90.522,Z 1258.628,A -85,B 0,C 180,E1 3228.327,E2 3228.327} C_VEL
LIN {X 0,Y 84.574,Z 1259.955,A -85,B 0,C 180,E1 3226.583,E2 3226.583} C_VEL
LIN {X 0,Y 61.03,Z 1264.567,A -85,B 0,C 180,E1 3212.302,E2 3212.302} C_VEL
LIN {X 0,Y 46.987,Z 1266.888,A -85,B 0,C 180,E1 3192.992,E2 3192.992} C_VEL
LIN {X 0,Y 40.68,Z 1267.992,A -85,B 0,C 180,E1 3168.701,E2 3168.701} C_VEL
LIN {X 0,Y 40.087,Z 1268.314,A -85,B 0,C 180,E1 3151.494,E2 3151.494} C_VEL
LIN {X 0,Y 40.221,Z 1268.101,A -85,B 0,C 180,E1 3137.139,E2 3137.139} C_VEL
LIN {X 0,Y 44.235,Z 1267.332,A -85,B 0,C 180,E1 3114.081,E2 3114.081} C_VEL
LIN {X 0,Y 55.912,Z 1265.408,A -85,B 0,C 180,E1 3092.898,E2 3092.898} C_VEL
LIN {X 0,Y 72.539,Z 1262.364,A -85,B 0,C 180,E1 3079.319,E2 3079.319} C_VEL
LIN {X 0,Y 91.552,Z 1258.233,A -85,B 0,C 180,E1 3070.771,E2 3070.771} C_VEL
LIN {X 0,Y 112.355,Z 1252.852,A -85,B 0,C 180,E1 3064.956,E2 3064.956} C_VEL
LIN {X 0,Y 138.931,Z 1244.669,A -85,B 0,C 180,E1 3060.142,E2 3060.142} C_VEL
LIN {X 0,Y 146.56,Z 1241.892,A -85,B 0,C 180,E1 3059.073,E2 3059.073} C_VEL
LIN {X 0,Y 124.314,Z 1248.919,A -85,B 0,C 180,E1 3055.514,E2 3055.514} C_VEL
LIN {X 0,Y 96.031,Z 1256.179,A -85,B 0,C 180,E1 3048.59,E2 3048.59} C_VEL
LIN {X 0,Y 75.471,Z 1260.331,A -85,B 0,C 180,E1 3040.05,E2 3040.05} C_VEL
LIN {X 0,Y 58.966,Z 1263.039,A -85,B 0,C 180,E1 3027.891,E2 3027.891} C_VEL
LIN {X 0,Y 46.729,Z 1264.711,A -85,B 0,C 180,E1 3009.618,E2 3009.618} C_VEL
LIN {X 0,Y 41.106,Z 1265.442,A -85,B 0,C 180,E1 2988.366,E2 2988.366} C_VEL
LIN {X 0,Y 40.103,Z 1265.697,A -85,B 0,C 180,E1 2969.935,E2 2969.935} C_VEL
LIN {X 0,Y 41.112,Z 1265.448,A -85,B 0,C 180,E1 2951.502,E2 2951.502} C_VEL
LIN {X 0,Y 47.307,Z 1264.658,A -85,B 0,C 180,E1 2928.993,E2 2928.993} C_VEL
LIN {X 0,Y 59.746,Z 1262.957,A -85,B 0,C 180,E1 2911.253,E2 2911.253} C_VEL
LIN {X 0,Y 77.4,Z 1260.035,A -85,B 0,C 180,E1 2898.842,E2 2898.842} C_VEL
LIN {X 0,Y 102.407,Z 1254.829,A -85,B 0,C 180,E1 2889.413,E2 2889.413} C_VEL
LIN {X 0,Y 126.335,Z 1248.401,A -85,B 0,C 180,E1 2884.023,E2 2884.023} C_VEL
LIN {X 0,Y 146.277,Z 1242.096,A -85,B 0,C 180,E1 2880.884,E2 2880.884} C_VEL
LIN {X 0,Y 122.186,Z 1250.108,A -85,B 0,C 180,E1 2877.061,E2 2877.061} C_VEL
LIN {X 0,Y 95.343,Z 1257.399,A -85,B 0,C 180,E1 2870.478,E2 2870.478} C_VEL
LIN {X 0,Y 84.574,Z 1259.955,A -85,B 0,C 180,E1 2866.583,E2 2866.583} C_VEL
LIN {X 0,Y 77.666,Z 1261.401,A -85,B 0,C 180,E1 2864.306,E2 2864.306} C_VEL
LIN {X 0,Y 57.134,Z 1264.437,A -85,B 0,C 180,E1 2858.466,E2 2858.466} C_VEL
LIN {X 0,Y 52.029,Z 1265.141,A -85,B 0,C 180,E1 2854.982,E2 2854.982} C_VEL
LIN {X 0,Y 37.066,Z 1267.206,A -85,B 0,C 180,E1 2830.946,E2 2830.946} C_VEL
LIN {X 0,Y 32.14,Z 1267.922,A -85,B 0,C 180,E1 2800.84,E2 2800.84} C_VEL
LIN {X 0,Y 32.084,Z 1268.024,A -85,B 0,C 180,E1 2786.508,E2 2786.508} C_VEL
LIN {X 0,Y 34.811,Z 1267.545,A -85,B 0,C 180,E1 2757.016,E2 2757.016} C_VEL
LIN {X 0,Y 49.556,Z 1265.504,A -85,B 0,C 180,E1 2727.525,E2 2727.525} C_VEL
LIN {X 0,Y 69.752,Z 1262.176,A -85,B 0,C 180,E1 2713.078,E2 2713.078} C_VEL
LIN {X 0,Y 90.359,Z 1257.956,A -85,B 0,C 180,E1 2705.523,E2 2705.523} C_VEL
LIN {X 0,Y 111.942,Z 1252.574,A -85,B 0,C 180,E1 2700.644,E2 2700.644} C_VEL
LIN {X 0,Y 121.635,Z 1249.872,A -85,B 0,C 180,E1 2698.999,E2 2698.999} C_VEL
LIN {X 0,Y 94.549,Z 1256.491,A -85,B 0,C 180,E1 2693.485,E2 2693.485} C_VEL
LIN {X 0,Y 73.059,Z 1260.604,A -85,B 0,C 180,E1 2686.175,E2 2686.175} C_VEL
LIN {X 0,Y 55.032,Z 1263.31,A -85,B 0,C 180,E1 2675.173,E2 2675.173} C_VEL
LIN {X 0,Y 40.86,Z 1264.97,A -85,B 0,C 180,E1 2657.136,E2 2657.136} C_VEL
LIN {X 0,Y 33.422,Z 1265.715,A -85,B 0,C 180,E1 2631.959,E2 2631.959} C_VEL
LIN {X 0,Y 32.106,Z 1265.959,A -85,B 0,C 180,E1 2609.919,E2 2609.919} C_VEL
LIN {X 0,Y 33.541,Z 1265.713,A -85,B 0,C 180,E1 2587.115,E2 2587.115} C_VEL
LIN {X 0,Y 41.488,Z 1264.926,A -85,B 0,C 180,E1 2561.568,E2 2561.568} C_VEL
LIN {X 0,Y 55.88,Z 1263.232,A -85,B 0,C 180,E1 2544.031,E2 2544.031} C_VEL
LIN {X 0,Y 74.931,Z 1260.34,A -85,B 0,C 180,E1 2532.924,E2 2532.924} C_VEL
LIN {X 0,Y 100.409,Z 1255.343,A -85,B 0,C 180,E1 2524.987,E2 2524.987} C_VEL
LIN {X 0,Y 121.479,Z 1250.008,A -85,B 0,C 180,E1 2520.943,E2 2520.943} C_VEL
LIN {X 0,Y 94.316,Z 1257.123,A -85,B 0,C 180,E1 2515.532,E2 2515.532} C_VEL
LIN {X 0,Y 72.564,Z 1261.694,A -85,B 0,C 180,E1 2508.213,E2 2508.213} C_VEL
LIN {X 0,Y 54.34,Z 1264.786,A -85,B 0,C 180,E1 2497.047,E2 2497.047} C_VEL
LIN {X 0,Y 52.029,Z 1265.141,A -85,B 0,C 180,E1 2494.982,E2 2494.982} C_VEL
LIN {X 0,Y 45.75,Z 1266.01,A -85,B 0,C 180,E1 2489.708,E2 2489.708} C_VEL
LIN {X 0,Y 27.547,Z 1267.386,A -85,B 0,C 180,E1 2467.023,E2 2467.023} C_VEL
LIN {X 0,Y 25.343,Z 1267.5,A -85,B 0,C 180,E1 2457.201,E2 2457.201} C_VEL
LIN {X 0,Y 24.098,Z 1267.804,A -85,B 0,C 180,E1 2430.109,E2 2430.109} C_VEL
LIN {X 0,Y 25.77,Z 1267.454,A -85,B 0,C 180,E1 2399.828,E2 2399.828} C_VEL
LIN {X 0,Y 37.358,Z 1266.258,A -85,B 0,C 180,E1 2368.119,E2 2368.119} C_VEL
LIN {X 0,Y 59.817,Z 1263.381,A -85,B 0,C 180,E1 2349.8,E2 2349.8} C_VEL
LIN {X 0,Y 85.955,Z 1258.548,A -85,B 0,C 180,E1 2341.062,E2 2341.062} C_VEL
LIN {X 0,Y 95.955,Z 1256.372,A -85,B 0,C 180,E1 2338.932,E2 2338.932} C_VEL
LIN {X 0,Y 72.488,Z 1260.726,A -85,B 0,C 180,E1 2332.967,E2 2332.967} C_VEL
LIN {X 0,Y 52.995,Z 1263.476,A -85,B 0,C 180,E1 2324.013,E2 2324.013} C_VEL
LIN {X 0,Y 36.535,Z 1265.178,A -85,B 0,C 180,E1 2307.899,E2 2307.899} C_VEL
LIN {X 0,Y 26.26,Z 1265.973,A -85,B 0,C 180,E1 2279.553,E2 2279.553} C_VEL
LIN {X 0,Y 24.117,Z 1266.204,A -85,B 0,C 180,E1 2252.267,E2 2252.267} C_VEL
LIN {X 0,Y 25.344,Z 1266.032,A -85,B 0,C 180,E1 2226.652,E2 2226.652} C_VEL
LIN {X 0,Y 33.759,Z 1265.438,A -85,B 0,C 180,E1 2196.774,E2 2196.774} C_VEL
LIN {X 0,Y 50.411,Z 1263.818,A -85,B 0,C 180,E1 2177.653,E2 2177.653} C_VEL
LIN {X 0,Y 69.699,Z 1261.213,A -85,B 0,C 180,E1 2167.924,E2 2167.924} C_VEL
LIN {X 0,Y 90.097,Z 1257.595,A -85,B 0,C 180,E1 2162.199,E2 2162.199} C_VEL
LIN {X 0,Y 95.801,Z 1256.464,A -85,B 0,C 180,E1 2161,E2 2161} C_VEL
LIN {X 0,Y 72.293,Z 1261.249,A -85,B 0,C 180,E1 2155.144,E2 2155.144} C_VEL
LIN {X 0,Y 51.665,Z 1264.513,A -85,B 0,C 180,E1 2145.578,E2 2145.578} C_VEL
LIN {X 0,Y 34.501,Z 1266.576,A -85,B 0,C 180,E1 2127.324,E2 2127.324} C_VEL
LIN {X 0,Y 25.343,Z 1267.5,A -85,B 0,C 180,E1 2097.201,E2 2097.201} C_VEL
LIN {X 0,Y 23.297,Z 1267.652,A -85,B 0,C 180,E1 2083.749,E2 2083.749} C_VEL
LIN {X 0,Y 20.708,Z 1267.659,A -85,B 0,C 180,E1 2064.447,E2 2064.447} C_VEL
LIN {X 0,Y 23.304,Z 1267.007,A -85,B 0,C 180,E1 2013.611,E2 2013.611} C_VEL
LIN {X 0,Y 25.682,Z 1266.766,A -85,B 0,C 180,E1 2007.699,E2 2007.699} C_VEL
LIN {X 0,Y 47.26,Z 1264.589,A -85,B 0,C 180,E1 1986.602,E2 1986.602} C_VEL
LIN {X 0,Y 69.181,Z 1261.416,A -85,B 0,C 180,E1 1978.869,E2 1978.869} C_VEL
LIN {X 0,Y 48.473,Z 1264.062,A -85,B 0,C 180,E1 1971.547,E2 1971.547} C_VEL
LIN {X 0,Y 29.539,Z 1265.69,A -85,B 0,C 180,E1 1955.831,E2 1955.831} C_VEL
LIN {X 0,Y 17.776,Z 1266.309,A -85,B 0,C 180,E1 1920.241,E2 1920.241} C_VEL
LIN {X 0,Y 16.129,Z 1266.471,A -85,B 0,C 180,E1 1886.284,E2 1886.284} C_VEL
LIN {X 0,Y 20.823,Z 1266.209,A -85,B 0,C 180,E1 1843.746,E2 1843.746} C_VEL
LIN {X 0,Y 41.282,Z 1264.898,A -85,B 0,C 180,E1 1812.591,E2 1812.591} C_VEL
LIN {X 0,Y 67.061,Z 1261.786,A -85,B 0,C 180,E1 1801.608,E2 1801.608} C_VEL
LIN {X 0,Y 69.022,Z 1261.489,A -85,B 0,C 180,E1 1801.089,E2 1801.089} C_VEL
LIN {X 0,Y 46.389,Z 1264.733,A -85,B 0,C 180,E1 1792.949,E2 1792.949} C_VEL
LIN {X 0,Y 23.651,Z 1266.978,A -85,B 0,C 180,E1 1767.931,E2 1767.931} C_VEL
LIN {X 0,Y 16.095,Z 1267.501,A -85,B 0,C 180,E1 1717.301,E2 1717.301} C_VEL
LIN {X 0,Y 16.197,Z 1267.443,A -85,B 0,C 180,E1 1695.871,E2 1695.871} C_VEL
LIN {X 0,Y 25.682,Z 1266.766,A -85,B 0,C 180,E1 1647.699,E2 1647.699} C_VEL
LIN {X 0,Y 25.943,Z 1266.653,A -85,B 0,C 180,E1 1643.813,E2 1643.813} C_VEL
LIN {X 0,Y 24.24,Z 1266.586,A -85,B 0,C 180,E1 1637.339,E2 1637.339} C_VEL
LIN {X 0,Y 20.176,Z 1266.646,A -85,B 0,C 180,E1 1627.825,E2 1627.825} C_VEL
LIN {X 0,Y 13.645,Z 1266.702,A -85,B 0,C 180,E1 1610.45,E2 1610.45} C_VEL
LIN {X 0,Y 8.549,Z 1266.761,A -85,B 0,C 180,E1 1571.469,E2 1571.469} C_VEL
LIN {X 0,Y 7.956,Z 1266.749,A -85,B 0,C 180,E1 1525.504,E2 1525.504} C_VEL
LIN {X 0,Y 8.675,Z 1266.683,A -85,B 0,C 180,E1 1506.274,E2 1506.274} C_VEL
LIN {X 0,Y 22.587,Z 1266.28,A -85,B 0,C 180,E1 1452.609,E2 1452.609} C_VEL
LIN {X 0,Y 39.673,Z 1265.215,A -85,B 0,C 180,E1 1441.19,E2 1441.19} C_VEL
LIN {X 0,Y 16.014,Z 1266.862,A -85,B 0,C 180,E1 1419.947,E2 1419.947} C_VEL
LIN {X 0,Y 8.093,Z 1267.279,A -85,B 0,C 180,E1 1350.323,E2 1350.323} C_VEL
LIN {X 0,Y 15.935,Z 1266.858,A -85,B 0,C 180,E1 1280.235,E2 1280.235} C_VEL
LIN {X 0,Y 39.958,Z 1265.168,A -85,B 0,C 180,E1 1258.705,E2 1258.705} C_VEL
LIN {X 0,Y 16.234,Z 1266.47,A -85,B 0,C 180,E1 1237.075,E2 1237.075} C_VEL
LIN {X 0,Y 8.156,Z 1266.729,A -85,B 0,C 180,E1 1176.719,E2 1176.719} C_VEL
LIN {X 0,Y 8.675,Z 1266.683,A -85,B 0,C 180,E1 1146.274,E2 1146.274} C_VEL
LIN {X 0,Y 7.666,Z 1266.725,A -85,B 0,C 180,E1 1142.409,E2 1142.409} C_VEL
LIN {X 0,Y 1.733,Z 1266.953,A -85,B 0,C 180,E1 1223.852,E2 1223.852} C_VEL
LIN {X 0,Y 1.226,Z 1266.987,A -85,B 0,C 180,E1 1257.272,E2 1257.272} C_VEL
LIN {X 0,Y 1.05,Z 1266.996,A -85,B 0,C 180,E1 1085.071,E2 1085.071} C_VEL
LIN {X 0,Y 1.226,Z 1266.987,A -85,B 0,C 180,E1 1257.272,E2 1257.272} C_VEL
LIN {X 0,Y 3.247,Z 1268.987,A -85,B 0,C 180,E1 1264.141,E2 1264.141} C_VEL
LIN {X 0,Y 3.247,Z 1292,A -85,B 0,C 180,E1 1264.141,E2 1264.141} C_VEL
LIN {X 0,Y 3.247,Z 1292,A -85,B 0,C 180,E1 1264.141,E2 1264.141}

QRS_NEXT_CUT()

QRS_NEXT()
QRS_HOME()

END
